RoboDK station: kr8_clean.rdk

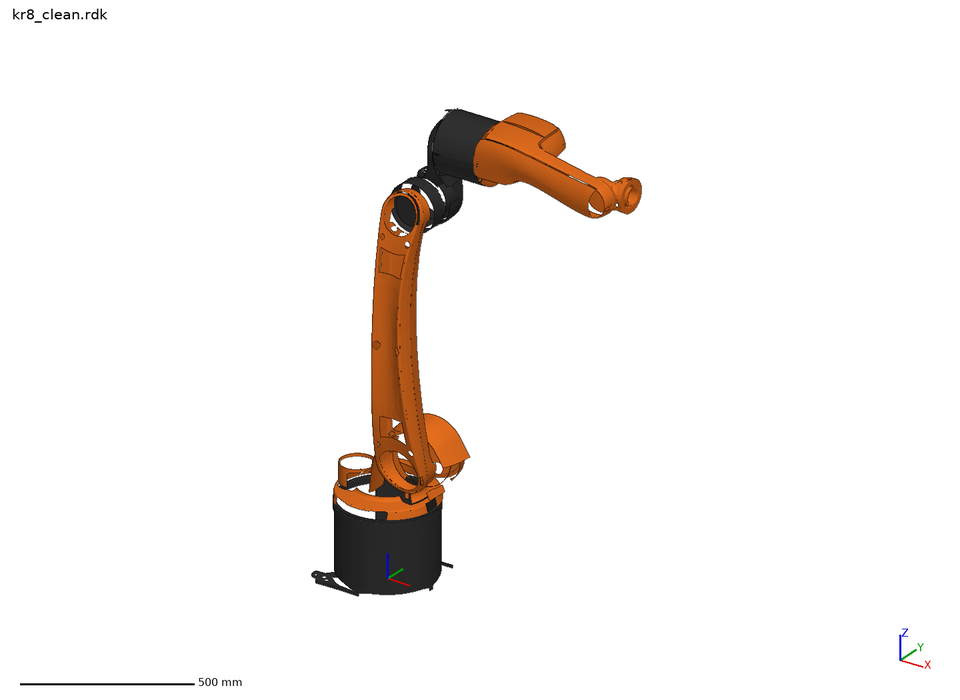
[picture v0: the station drawn from its stored meshes, robots at their saved joint values, targets as dots, program paths as lines]
Station kr8_clean (saved by RoboDK 5.1.0). Poses are relative to the parent item; angles as X-Y-Z fixed-axis rotations.
  - frame KR 8 1620 ARC HW Base at (0, 0, 0) mm
    - robot KR 8 1620 ARC HW: 6 axes
        modified DH rows (alpha deg, a mm, theta deg, d mm): 0, 0, 0, 450; -90, 150, 0, 0; 0, 810, -90, 0; -90, 200, 0, 630; 90, 0, 0, 0; -90, 0, 180, 80
        joint limits [-170, -185, -120, -165, -115, -350] to [170, 65, 180, 165, 140, 350]; home [0, -90, 90, 0, 0, 0]; saved at [0, -90, 90, 0, 0, 0]
